{attribute 'GeneratedUsingTerminal: KL6224-0003'}
{attribute addProperty BoxType "KL6224-0003"}
{attribute addProperty Description ""}
{attribute addProperty Physics ""}
{attribute addProperty Id "Channel_1AT %Q*Channel_779103830"}
{attribute addProperty CRC "2126695780"}
{attribute addProperty Size "0"}
TYPE KL_7EC2CD64 :
STRUCT
	{attribute addProperty Name "Channel_1"}
	Channel_1 : Channel_77910383;
END_STRUCT
END_TYPE

(* stored: Version 1.2.0.0, ProductVersion 3.1.4024.11
   DUT KL_7EC2CD64: Id {e703fc5a-4e0f-4104-a965-70a55e7bca9d} *)
